TYPE ST_HMI_DataSourceHistRecordInfo : 
STRUCT
	nID: DINT;
	sName: WSTRING(80);
	sDisplayName: WSTRING(80);
	dtRecordStart: DCTIMESTRUCT;
	dtRecordEnd: DCTIMESTRUCT;
	dtSelectedRangeStart: DCTIMESTRUCT;
	dtSelectedRangeEnd: DCTIMESTRUCT;
END_STRUCT
END_TYPE

(* stored: DUT ST_HMI_DataSourceHistRecordInfo: Id 7c58b423-57c5-4f0f-87ec-3bde51983792 *)
